FUNCTION_BLOCK "G099M_Code"
TITLE =G099M COUPLING DEVICE WALL GERM 1
//COPYRIGHT:    (C) 2009  BUHLER AG, CH-9240 UZWIL, SWITZERLAND
//
//PRODUCT:      WinCoS_BIW01_09
//
//TITLE:        COUPLING DEVICE WALL GERM 1
//                Machine group control
//                Maschinengruppensteuerung
//
//--------------------------------------------------------------------------------
//
//IDENT:        AUTHOR:             DEPT:                              DATE:
//
//P01_FB199.1.0 K.Renz              CSB41                              29.Sep.2009
//             1st Release
//
//--------------------------------------------------------------------------------
//
//PURPOSE:
//
//MANUAL :
//
//RESTRICTIONS:
//
//--------------------------------------------------------------------------------
AUTHOR : KR
FAMILY : USW
VERSION : 9.9


VAR
  Gr : "GCS7_GrpCtrlSub";	//Standard interface to group
  InOutValue1 : DINT ;	//Data for user
  InOutValue2 : DINT ;	//Data for user
  OutWayConflict : BOOL ;	//Data for user
  OutSelectionOk : BOOL ;	//Data for user
  CmdNewValue : BOOL ;	//Data for user
  CmdNewJob : BOOL ;	//Data for user
  OutCodeOK : BOOL ;	//Data for user
  InEndOfJob : BOOL ;	//Data for user
  staWayOk : BOOL ;	//Data for user
  EdgeStartRelease : BOOL ;	//Data for user
  USW8 : BOOL ;	//Data for user
  USW9 : BOOL ;	//Data for user
  USW10 : BOOL ;	//Data for user
  USW11 : BOOL ;	//Data for user
  USW12 : BOOL ;	//Data for user
  USW13 : BOOL ;	//Data for user
  USW14 : BOOL ;	//Data for user
  USW15 : BOOL ;	//Data for user
  A_2115_BZS42 : "GCS7_E_DigInput";	// DigInpCont
  A_2115_BZS43 : "GCS7_E_DigInput";	// DigInpCont
  A_2115_BZS46 : "GCS7_E_DigInput";	// DigInpCont
  A_2115_BZS47 : "GCS7_E_DigInput";	// DigInpCont
  A_2115_MXZ41 : "GCS7_E_Motor";	// Motor
  A_2115_MXZ45 : "GCS7_E_Motor";	// Motor
END_VAR
VAR_TEMP
  tmpEnable : BOOL ;
  tmpFlag : BOOL ;
  tmpCmdNext : BOOL ;
  tmpLocal : BOOL ;
  tmpAspOk : BOOL ;
  tmpHWStop : BOOL ;
  tmpInstanzDBNo : INT ;
END_VAR
BEGIN
NETWORK
TITLE =



NETWORK
TITLE =Read command from group control
//Parameter
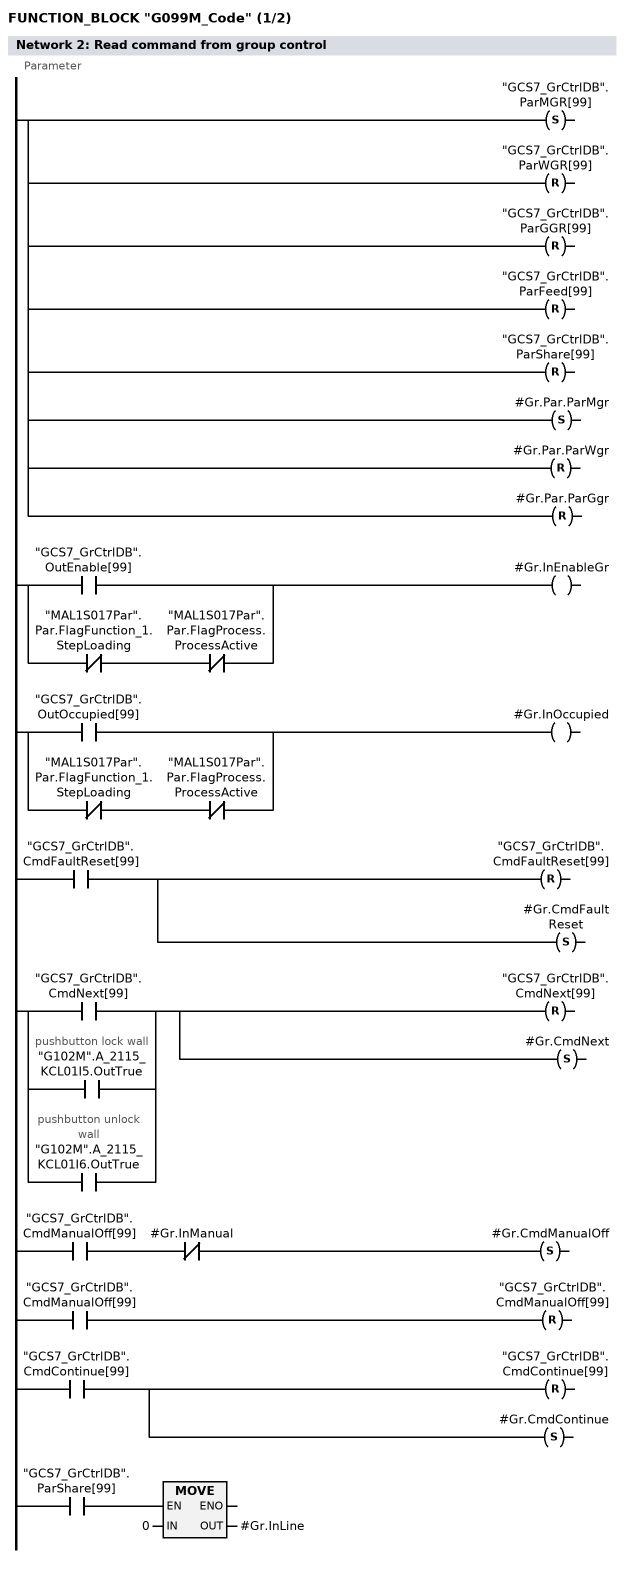
      SET   ;
      S     "GCS7_GrCtrlDB".ParMGR[99];
      R     "GCS7_GrCtrlDB".ParWGR[99];
      R     "GCS7_GrCtrlDB".ParGGR[99];
      R     "GCS7_GrCtrlDB".ParFeed[99];
      R     "GCS7_GrCtrlDB".ParShare[99];
      S     #Gr.Par.ParMgr;
      R     #Gr.Par.ParWgr;
      R     #Gr.Par.ParGgr;
//Command
      U     "GCS7_GrCtrlDB".OutEnable[99];
      O(    ;
      UN    "MAL1S017Par".Par.FlagFunction_1.StepLoading;
      UN    "MAL1S017Par".Par.FlagProcess.ProcessActive;
      )     ;
      =     #Gr.InEnableGr;
      U     "GCS7_GrCtrlDB".OutOccupied[99];
      O(    ;
      UN    "MAL1S017Par".Par.FlagFunction_1.StepLoading;
      UN    "MAL1S017Par".Par.FlagProcess.ProcessActive;
      )     ;
      =     #Gr.InOccupied;
      U     "GCS7_GrCtrlDB".CmdFaultReset[99];
      R     "GCS7_GrCtrlDB".CmdFaultReset[99];
      S     #Gr.CmdFaultReset;
      U     "GCS7_GrCtrlDB".CmdNext[99];
      O     "G102M".A_2115_KCL01I5.OutTrue; // pushbutton lock wall
      O     "G102M".A_2115_KCL01I6.OutTrue; // pushbutton unlock wall
      R     "GCS7_GrCtrlDB".CmdNext[99];
      S     #Gr.CmdNext;

      U     "GCS7_GrCtrlDB".CmdManualOff[99];
      UN    #Gr.InManual;
//JV020310      SET                               // No PC-Direct-Controll!!!
      S     #Gr.CmdManualOff;
      U     "GCS7_GrCtrlDB".CmdManualOff[99];
      R     "GCS7_GrCtrlDB".CmdManualOff[99];

//      U     "GCS7_GrCtrlDB".CmdManualOff[99]
//      O     "GCS7_GrCtrlDB".OutOccupied[99]
//      R     "GCS7_GrCtrlDB".CmdManualOff[99]
//      S     #Gr.CmdManualOff

      U     "GCS7_GrCtrlDB".CmdContinue[99];
      R     "GCS7_GrCtrlDB".CmdContinue[99];
      S     #Gr.CmdContinue;
//Init Line Number
      U     "GCS7_GrCtrlDB".ParShare[99];
      SPBN  WE00;
      L     0;
      T     #Gr.InLine;
WE00: NOP   0;
NETWORK
TITLE =Call Methode Control
// 1. Handle Interface PCControl
// 2. Prepare mode --> ModePassive,ModeActive,ModeIdling
// 3. Reset global flags of the group
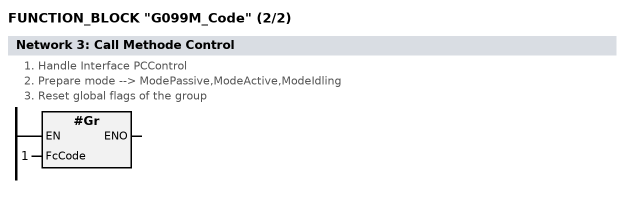
      CALL #Gr (
           FcCode                   := 1);
NETWORK
TITLE =Restart Idling Time

      L     #Gr.Par.ParIdling;
      L     2;
      >=I   ;
      SPB   IdTm;
      T     #Gr.Par.ParIdling;
IdTm: NOP   0;
      CLR   ;
      S     #Gr.CmdRestartIdling;
NETWORK
TITLE =Prepare global flags



NETWORK
TITLE =Set Pattern (Target position)



NETWORK
TITLE =Interlocking WayOk
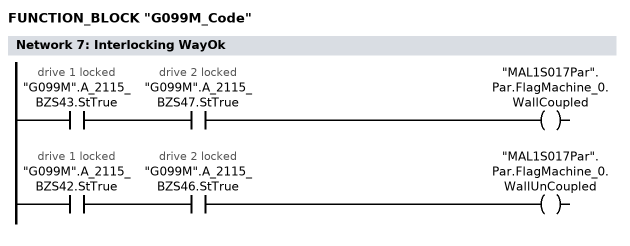

      U     "G099M".A_2115_BZS43.StTrue; // drive 1 locked
      U     "G099M".A_2115_BZS47.StTrue; // drive 2 locked
      =     "MAL1S017Par".Par.FlagMachine_0.WallCoupled;


      U     "G099M".A_2115_BZS42.StTrue; // drive 1 locked
      U     "G099M".A_2115_BZS46.StTrue; // drive 2 locked
      =     "MAL1S017Par".Par.FlagMachine_0.WallUnCoupled;

NETWORK
TITLE =Interlocking Autostart

      CLR   ;
      R     #Gr.OutAutostart;
NETWORK
TITLE =Interlocking Enable
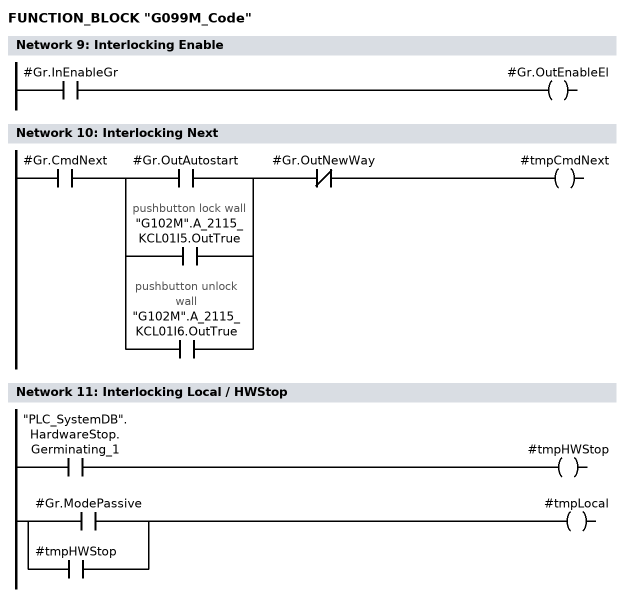

      U     #Gr.InEnableGr;
      =     #Gr.OutEnableEl;

NETWORK
TITLE =Interlocking Next

      U     #Gr.CmdNext;
      U(    ;
      U     #Gr.OutAutostart;
      O     "G102M".A_2115_KCL01I5.OutTrue; // pushbutton lock wall
      O     "G102M".A_2115_KCL01I6.OutTrue; // pushbutton unlock wall
      )     ;
      UN    #Gr.OutNewWay;
      =     #tmpCmdNext;

NETWORK
TITLE =Interlocking Local / HWStop

      U     "PLC_SystemDB".HardwareStop.Germinating_1;
      =     #tmpHWStop;

      U     #Gr.ModePassive;
      O     #tmpHWStop;
      =     #tmpLocal;

NETWORK
TITLE ==A-2115-BZS42 : COUPLING DRIVE UNLOCKED

      NOP   0;
//-InLocal---
      U     #tmpLocal;
      =     #A_2115_BZS42.InLocal;
//
//-Monitoring---
      U     "MAL1S017Par".Par.FlagFunction_1.StepUnloading; // Step unloading
      O     "MAL1S017Par".Par.FlagFunction_1.StepCleaning; // Step cleaning
      UN    #A_2115_BZS42.InpTrue;
      =     #A_2115_BZS42.InMonTrue;
      CLR   ;
      =     #A_2115_BZS42.InMonFalse;
//
//-PreAlarm---
      CLR   ;
      =     #A_2115_BZS42.InPreAlarmTrue;
      CLR   ;
      =     #A_2115_BZS42.InPreAlarmFalse;
//
//-Additional commands---
//      CLR
//      S     #A_2115_BZS42.CmdRunTimeOutTime
//
//-Read inputs---
      U     "A_2115_BZS42_I1";
      =     #A_2115_BZS42.InpTrue;
      U     "PLC_SystemDB".HardwareStop.Germinating_1;
      =     #A_2115_BZS42.InHWStop;
      U     "PLC_DPInfo".Master[1].SlavesError[15];
      =     #A_2115_BZS42.InDPFault;
//
//-Set Parameters---
//
//-Call object control---
      CALL #A_2115_BZS42 ;
//
//-Write outputs---
NETWORK
TITLE ==A-2115-BZS43 : COUPLING DRIVE LOCKED

      NOP   0;
//-InLocal---
      U     #tmpLocal;
      =     #A_2115_BZS43.InLocal;
//
//-Monitoring---
      U     "MAL1S017Par".Par.FlagFunction_1.StepLoading;
      O     "MAL1S017Par".Par.FlagProcess.ProcessActive;
      UN    #A_2115_BZS43.InpTrue;
      =     #A_2115_BZS43.InMonTrue;
      CLR   ;
      =     #A_2115_BZS43.InMonFalse;
//
//-PreAlarm---
      CLR   ;
      =     #A_2115_BZS43.InPreAlarmTrue;
      CLR   ;
      =     #A_2115_BZS43.InPreAlarmFalse;
//
//-Additional commands---
//      CLR
//      S     #A_2115_BZS43.CmdRunTimeOutTime
//
//-Read inputs---
      U     "A_2115_BZS43_I1";
      =     #A_2115_BZS43.InpTrue;
      U     "PLC_SystemDB".HardwareStop.Germinating_1;
      =     #A_2115_BZS43.InHWStop;
      U     "PLC_DPInfo".Master[1].SlavesError[15];
      =     #A_2115_BZS43.InDPFault;
//
//-Set Parameters---
//
//-Call object control---
      CALL #A_2115_BZS43 ;
//
//-Write outputs---
NETWORK
TITLE ==A-2115-BZS46 : COUPLING DRIVE UNLOCKED

      NOP   0;
//-InLocal---
      U     #tmpLocal;
      =     #A_2115_BZS46.InLocal;
//
//-Monitoring---
      U     "MAL1S017Par".Par.FlagFunction_1.StepUnloading; // Step unloading
      O     "MAL1S017Par".Par.FlagFunction_1.StepCleaning; // Step cleaning
      UN    #A_2115_BZS46.InpTrue;
      =     #A_2115_BZS46.InMonTrue;
      CLR   ;
      =     #A_2115_BZS46.InMonFalse;
//
//-PreAlarm---
      CLR   ;
      =     #A_2115_BZS46.InPreAlarmTrue;
      CLR   ;
      =     #A_2115_BZS46.InPreAlarmFalse;
//
//-Additional commands---
//      CLR
//      S     #A_2115_BZS46.CmdRunTimeOutTime
//
//-Read inputs---
      U     "A_2115_BZS46_I1";
      =     #A_2115_BZS46.InpTrue;
      U     "PLC_SystemDB".HardwareStop.Germinating_1;
      =     #A_2115_BZS46.InHWStop;
      U     "PLC_DPInfo".Master[1].SlavesError[15];
      =     #A_2115_BZS46.InDPFault;
//
//-Set Parameters---
//
//-Call object control---
      CALL #A_2115_BZS46 ;
//
//-Write outputs---
NETWORK
TITLE ==A-2115-BZS47 : COUPLING DRIVE LOCKED

      NOP   0;
//-InLocal---
      U     #tmpLocal;
      =     #A_2115_BZS47.InLocal;
//
//-Monitoring---
      U     "MAL1S017Par".Par.FlagFunction_1.StepLoading;
      O     "MAL1S017Par".Par.FlagProcess.ProcessActive;
      UN    #A_2115_BZS47.InpTrue;
      =     #A_2115_BZS47.InMonTrue;
      CLR   ;
      =     #A_2115_BZS47.InMonFalse;
//
//-PreAlarm---
      CLR   ;
      =     #A_2115_BZS47.InPreAlarmTrue;
      CLR   ;
      =     #A_2115_BZS47.InPreAlarmFalse;
//
//-Additional commands---
//      CLR
//      S     #A_2115_BZS47.CmdRunTimeOutTime
//
//-Read inputs---
      U     "A_2115_BZS47_I1";
      =     #A_2115_BZS47.InpTrue;
      U     "PLC_SystemDB".HardwareStop.Germinating_1;
      =     #A_2115_BZS47.InHWStop;
      U     "PLC_DPInfo".Master[1].SlavesError[15];
      =     #A_2115_BZS47.InDPFault;
//
//-Set Parameters---
//
//-Call object control---
      CALL #A_2115_BZS47 ;
//
//-Write outputs---
NETWORK
TITLE ==A-2115-MXZ41 : WALL COUPLING DRIVE
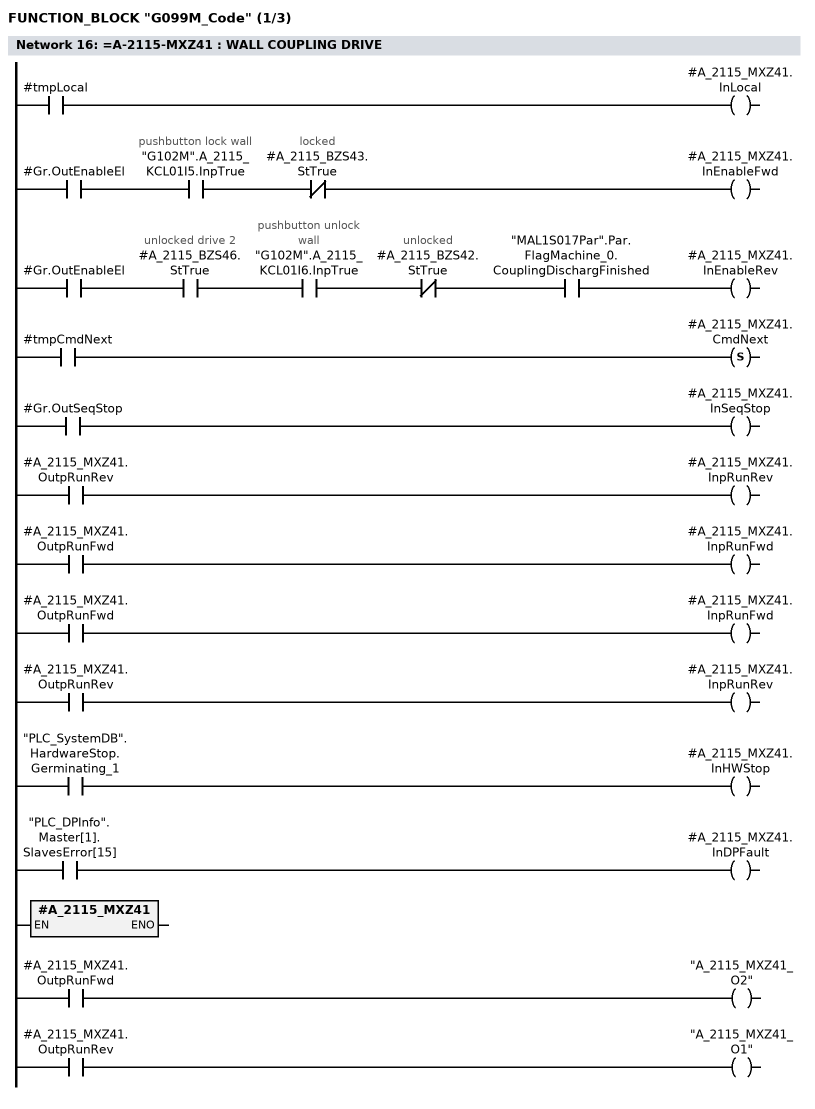

      NOP   0;
//-InLocal---
      U     #tmpLocal;
      =     #A_2115_MXZ41.InLocal;
//
//-Interlocking---
      U     #Gr.OutEnableEl;
      U     "G102M".A_2115_KCL01I5.InpTrue; // pushbutton lock wall
      UN    #A_2115_BZS43.StTrue; // locked
      =     #A_2115_MXZ41.InEnableFwd;
      U     #Gr.OutEnableEl;
      U     #A_2115_BZS46.StTrue; // unlocked drive 2
      U     "G102M".A_2115_KCL01I6.InpTrue; // pushbutton unlock wall
      UN    #A_2115_BZS42.StTrue; // unlocked
      U     "MAL1S017Par".Par.FlagMachine_0.CouplingDischargFinished;
      =     #A_2115_MXZ41.InEnableRev;
//
      U     #tmpCmdNext;
      S     #A_2115_MXZ41.CmdNext;
//
      U     #Gr.OutSeqStop;
      =     #A_2115_MXZ41.InSeqStop;
//
//-Read inputs---
      U     #A_2115_MXZ41.OutpRunRev;
      =     #A_2115_MXZ41.InpRunRev;
      U     #A_2115_MXZ41.OutpRunFwd;
      =     #A_2115_MXZ41.InpRunFwd;
      U     #A_2115_MXZ41.OutpRunFwd;
      =     #A_2115_MXZ41.InpRunFwd;
      U     #A_2115_MXZ41.OutpRunRev;
      =     #A_2115_MXZ41.InpRunRev;
      U     "PLC_SystemDB".HardwareStop.Germinating_1;
      =     #A_2115_MXZ41.InHWStop;
      U     "PLC_DPInfo".Master[1].SlavesError[15];
      =     #A_2115_MXZ41.InDPFault;
//
//-Set Parameters---
//
//-Call object control---
      CALL #A_2115_MXZ41 ;
//
//-Write outputs---
      U     #A_2115_MXZ41.OutpRunFwd;
      =     "A_2115_MXZ41_O2";
      U     #A_2115_MXZ41.OutpRunRev;
      =     "A_2115_MXZ41_O1";
NETWORK
TITLE ==A-2115-MXZ45 : WALL COUPLING DRIVE
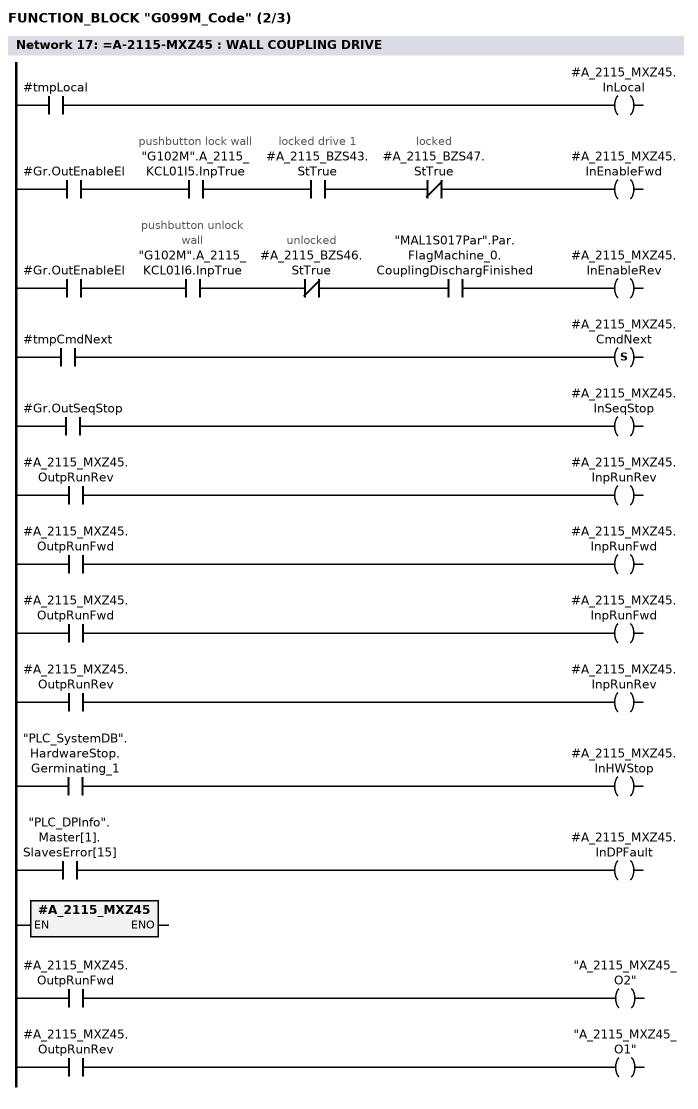

      NOP   0;
//-InLocal---
      U     #tmpLocal;
      =     #A_2115_MXZ45.InLocal;
//
//-Interlocking---
      U     #Gr.OutEnableEl;
      U     "G102M".A_2115_KCL01I5.InpTrue; // pushbutton lock wall
      U     #A_2115_BZS43.StTrue; // locked drive 1
      UN    #A_2115_BZS47.StTrue; // locked
      =     #A_2115_MXZ45.InEnableFwd;
      U     #Gr.OutEnableEl;
      U     "G102M".A_2115_KCL01I6.InpTrue; // pushbutton unlock wall
      UN    #A_2115_BZS46.StTrue; // unlocked
      U     "MAL1S017Par".Par.FlagMachine_0.CouplingDischargFinished;
      =     #A_2115_MXZ45.InEnableRev;
//
      U     #tmpCmdNext;
      S     #A_2115_MXZ45.CmdNext;
//
      U     #Gr.OutSeqStop;
      =     #A_2115_MXZ45.InSeqStop;
//
//-Read inputs---
      U     #A_2115_MXZ45.OutpRunRev;
      =     #A_2115_MXZ45.InpRunRev;
      U     #A_2115_MXZ45.OutpRunFwd;
      =     #A_2115_MXZ45.InpRunFwd;
      U     #A_2115_MXZ45.OutpRunFwd;
      =     #A_2115_MXZ45.InpRunFwd;
      U     #A_2115_MXZ45.OutpRunRev;
      =     #A_2115_MXZ45.InpRunRev;
      U     "PLC_SystemDB".HardwareStop.Germinating_1;
      =     #A_2115_MXZ45.InHWStop;
      U     "PLC_DPInfo".Master[1].SlavesError[15];
      =     #A_2115_MXZ45.InDPFault;
//
//-Set Parameters---
//
//-Call object control---
      CALL #A_2115_MXZ45 ;
//
//-Write outputs---
      U     #A_2115_MXZ45.OutpRunFwd;
      =     "A_2115_MXZ45_O2";
      U     #A_2115_MXZ45.OutpRunRev;
      =     "A_2115_MXZ45_O1";
NETWORK
TITLE =Test Fault
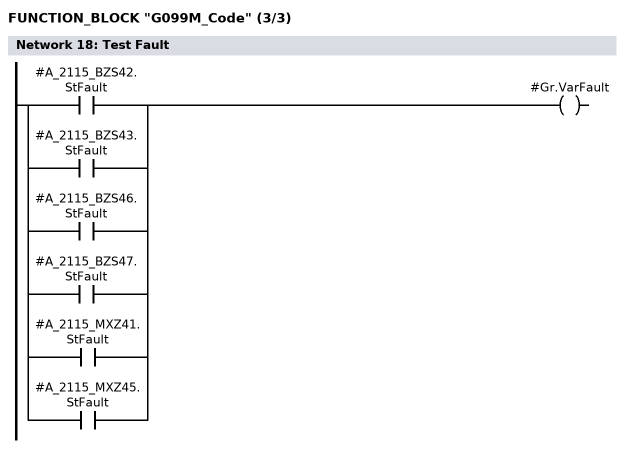

      U     #A_2115_BZS42.StFault;
      O     #A_2115_BZS43.StFault;
      O     #A_2115_BZS46.StFault;
      O     #A_2115_BZS47.StFault;
      O     #A_2115_MXZ41.StFault;
      O     #A_2115_MXZ45.StFault;
      =     #Gr.VarFault;
NETWORK
TITLE =Test Warning

      CLR   ;
      =     #Gr.OutWarning;
NETWORK
TITLE =Test Stopped
//      U     #A_2115_MXZ41.StStopped
//      U     #A_2115_MXZ45.StStopped
//
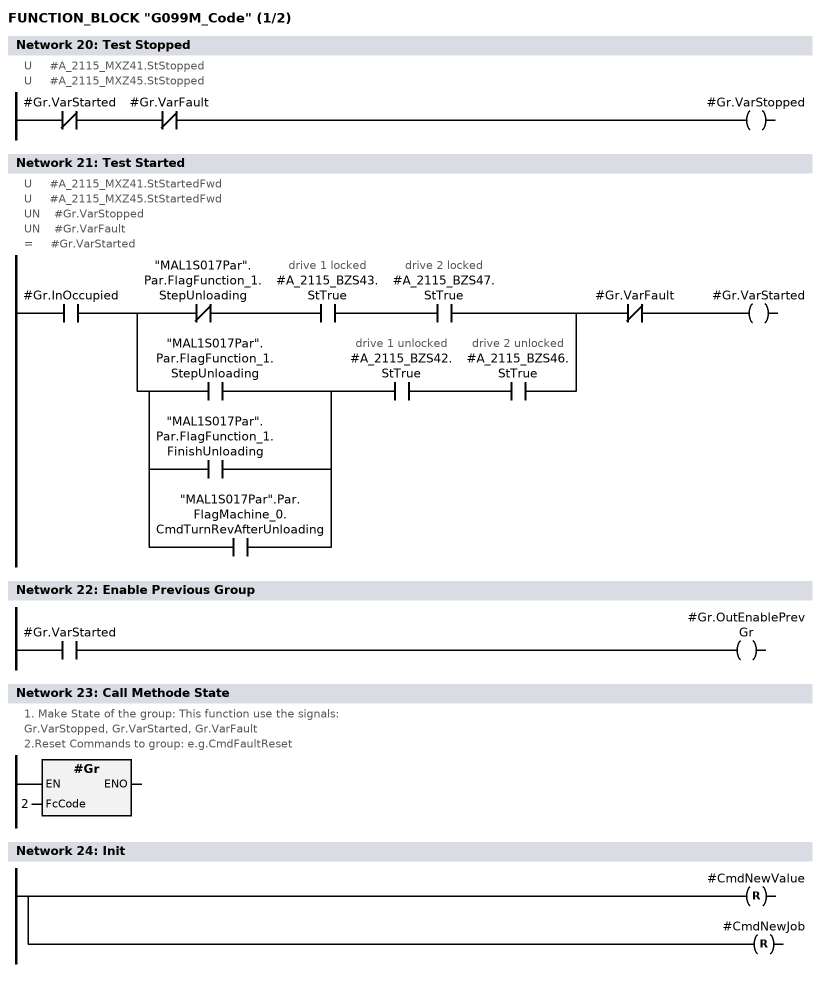
      UN    #Gr.VarStarted;
      UN    #Gr.VarFault;
      =     #Gr.VarStopped;
NETWORK
TITLE =Test Started
//      U     #A_2115_MXZ41.StStartedFwd
//      U     #A_2115_MXZ45.StStartedFwd
//      UN    #Gr.VarStopped
//      UN    #Gr.VarFault
//      =     #Gr.VarStarted
//
      U     #Gr.InOccupied;
      U(    ;
      O(    ;
      UN    "MAL1S017Par".Par.FlagFunction_1.StepUnloading;
      U     #A_2115_BZS43.StTrue; // drive 1 locked
      U     #A_2115_BZS47.StTrue; // drive 2 locked
      )     ;
      O(    ;
      U     "MAL1S017Par".Par.FlagFunction_1.StepUnloading;
      O     "MAL1S017Par".Par.FlagFunction_1.FinishUnloading;
      O     "MAL1S017Par".Par.FlagMachine_0.CmdTurnRevAfterUnloading;
      U     #A_2115_BZS42.StTrue; // drive 1 unlocked
      U     #A_2115_BZS46.StTrue; // drive 2 unlocked
      )     ;
      )     ;
      UN    #Gr.VarFault;
      =     #Gr.VarStarted;
NETWORK
TITLE =Enable Previous Group

      U     #Gr.VarStarted;
      =     #Gr.OutEnablePrevGr;
NETWORK
TITLE =Call Methode State
//1. Make State of the group: This function use the signals:
//        Gr.VarStopped, Gr.VarStarted, Gr.VarFault
//2.Reset Commands to group: e.g.CmdFaultReset
      CALL #Gr (
           FcCode                   := 2);
NETWORK
TITLE =Init

      SET   ;
      R     #CmdNewValue;
      R     #CmdNewJob;
NETWORK
TITLE =Write data to group control
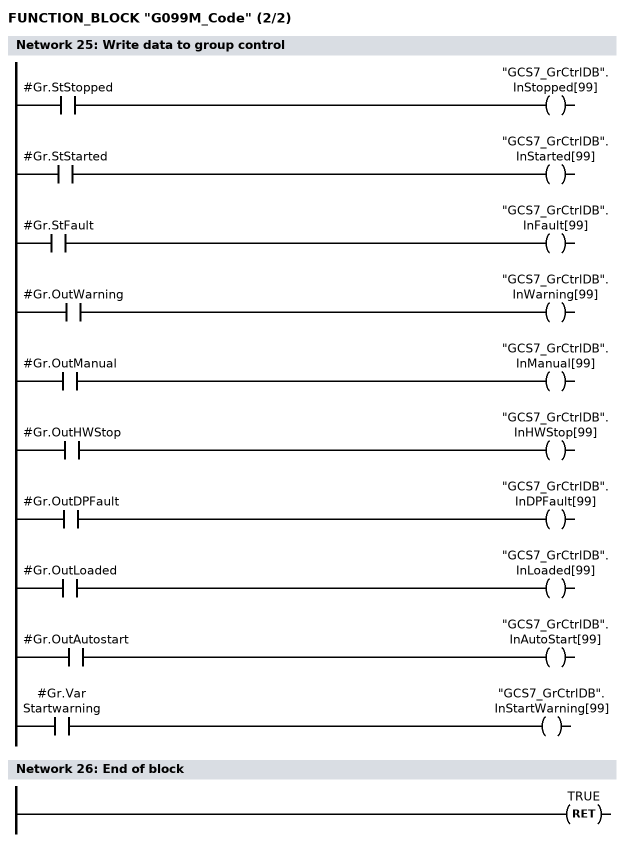

      U     #Gr.StStopped;
      =     "GCS7_GrCtrlDB".InStopped[99];
      U     #Gr.StStarted;
      =     "GCS7_GrCtrlDB".InStarted[99];
      U     #Gr.StFault;
      =     "GCS7_GrCtrlDB".InFault[99];
      U     #Gr.OutWarning;
      =     "GCS7_GrCtrlDB".InWarning[99];
      U     #Gr.OutManual;
      =     "GCS7_GrCtrlDB".InManual[99];
      U     #Gr.OutHWStop;
      =     "GCS7_GrCtrlDB".InHWStop[99];
      U     #Gr.OutDPFault;
      =     "GCS7_GrCtrlDB".InDPFault[99];
      U     #Gr.OutLoaded;
      =     "GCS7_GrCtrlDB".InLoaded[99];
      U     #Gr.OutAutostart;
      =     "GCS7_GrCtrlDB".InAutoStart[99];
      U     #Gr.VarStartwarning;
      =     "GCS7_GrCtrlDB".InStartWarning[99];
NETWORK
TITLE =End of block

      BE    ;

END_FUNCTION_BLOCK

